// TIA Portal V17 export
// export: Created 2024-09-02T12:50:01.5701323Z, ExportSetting WithDefaults, DisplayName Totally Integrated Automation Portal, DisplayVersion V17, DisplayName TIA Portal Openness, DisplayVersion V17, DisplayName TIA Portal Version Control Interface, DisplayVersion V17, DisplayName STEP 7 Professional, DisplayVersion V17, DisplayName STEP 7 Safety, DisplayVersion V17, DisplayName WinCC Professional, DisplayVersion V17
FUNCTION_BLOCK "GraFB_Hand_51_58"   // FB1175, GRAPH
TITLE = GRAPH FB
AUTHOR : OlegFuehrus
FAMILY : SK
NAME : SK
VERSION : 0.1
// Hand functions / Handfunktionen
// stored: AcknowledgeErrorsRequired true, AutoNumber true, ExtensionBlockName LTLL_ManualGraphExt, GraphVersion 4.0, InitialValuesAcquisition false, IsIECCheckEnabled false, LanguageInNetworks LAD, LockOperatingMode false, PermanentILProcessingInMANMode true, SetENOAutomatically false, SkipSteps false, UDAEnableTagReadback false, WithAlarmHandling true
   // inherited from GRAPH_BASE
   VAR
      OFF_SQ_BASE : Bool;
   END_VAR
   VAR_INPUT
      OFF_SQ : Bool;
      INIT_SQ : Bool;
      ACK_EF : Bool;
      S_PREV : Bool;
      S_NEXT : Bool;
      SW_AUTO : Bool;
      SW_TAP : Bool;
      SW_MAN : Bool;
      S_SEL : Int;
      S_ON : Bool;
      S_OFF : Bool;
      T_PUSH : Bool;
   END_VAR
   VAR_OUTPUT
      S_NO : Int;
      S_MORE : Bool;
      S_ACTIVE : Bool;
      ERR_FLT : Bool;
      AUTO_ON : Bool;
      TAP_ON : Bool;
      MAN_ON : Bool;
   END_VAR
   VAR
      extBlock { S7_SetPoint := 'True'} : "LTLL_ManualGraphExt";
   END_VAR
   VAR_TEMP
      t_FrgHand : Bool;   // Freigabe Handbetrieb / Enable manual operation
      t_Service : Bool;   // Servicebetrieb aktiv / Service operation active
   END_VAR
BEGIN
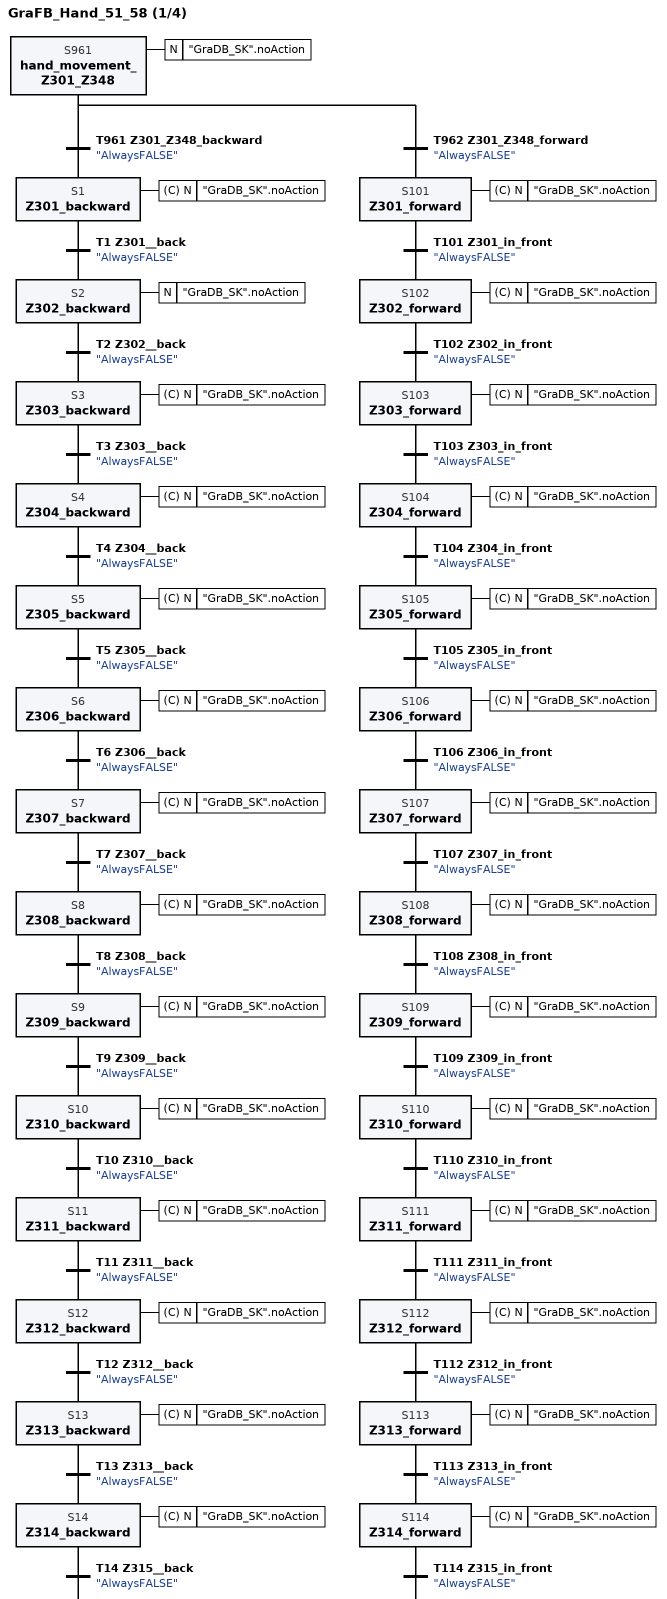
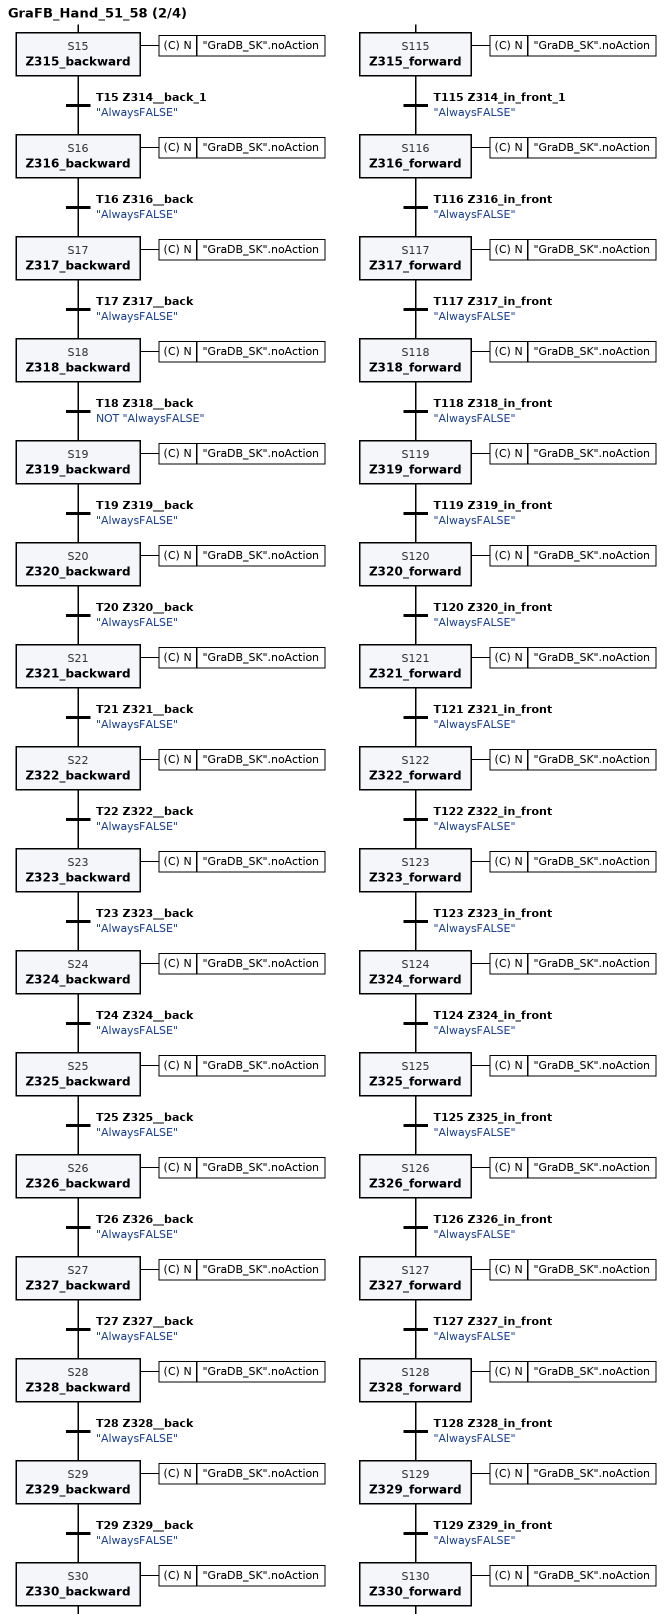
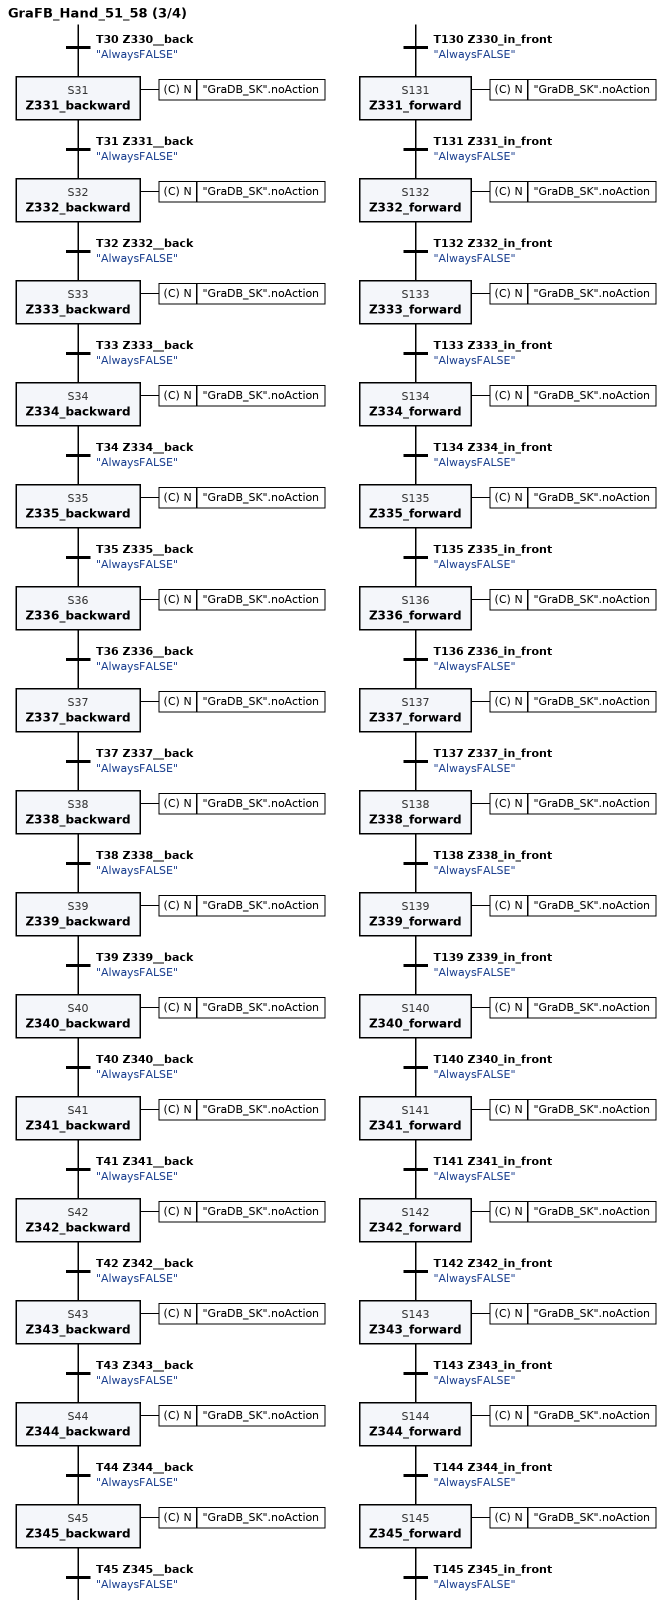
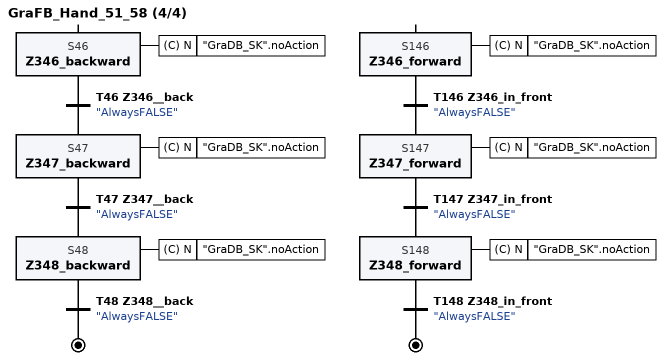
   // permanent pre-instructions
   NETWORK 1
   TITLE = HMI Lite Pass on data / HMI Lite Daten weiterreichen
      #extBlock.input := "LTLL_ManualGraphControl_OP70".screen[0].input;
   NETWORK 2
   TITLE = Instance DB Name query and pass on / Instanz DB Name abfragen und weiterreichen
      GetInstanceName(size := 0, OUT => #extBlock.input.instanceName);
   NETWORK 3
   TITLE = Interlocks Permanent machining, manual Approve and service / Interlocks Permanent Bearbeiten, Handfreigabe und Service
      IF NOT #RT_DATA.MOP.IL_PERM THEN #RT_DATA.MOP.IL_PERM := TRUE; END_IF;
      #t_FrgHand := "AnwDB_OperatingModes_OP70".BA[0]."mode_hand+start";
      #t_Service := "AnwDB_OperatingModes_OP70".BA[0].mode_service;

   // sequencer 1: Sequencer 1
   STEP hand_movement_Z301_Z348:   // S961, max time T#10S, warning time T#7S: Step commentary / Schrittkommentar
      interlock C := (none);   // hand_bereich_Z001_Z005
      supervision V := (none);   // hand_bereich_Z001_Z005
              N    "GraDB_SK".noAction
   END_STEP
   TRANSITION Z301_Z348_backward FROM hand_movement_Z301_Z348 TO Z301_backward   // T961
      := "AlwaysFALSE";
   END_TRANSITION
   TRANSITION Z301_Z348_forward FROM hand_movement_Z301_Z348 TO Z301_forward   // T962
      := "AlwaysFALSE";
   END_TRANSITION
   STEP Z301_backward:   // S1, max time T#10S, warning time T#7S
      interlock C := "AlwaysFALSE";   // Z301_zur
      supervision V := NOT #Z301__back.TT AND (#Z301_backward.T > T#5S);   // Z301_zur
      (C)     N    "GraDB_SK".noAction
   END_STEP
   TRANSITION Z301__back FROM Z301_backward TO Z302_backward   // T1
      := "AlwaysFALSE";
   END_TRANSITION
   STEP Z302_backward:   // S2, max time T#10S, warning time T#7S
      interlock C := "AlwaysFALSE";   // Z302_zur
      supervision V := NOT #Z302__back.TT AND (#Z302_backward.T > T#5S);   // Z302_zur
              N    "GraDB_SK".noAction
   END_STEP
   TRANSITION Z302__back FROM Z302_backward TO Z303_backward   // T2
      := "AlwaysFALSE";
   END_TRANSITION
   STEP Z303_backward:   // S3, max time T#10S, warning time T#7S
      interlock C := "AlwaysFALSE";   // Z303_zur
      supervision V := NOT #Z303__back.TT AND (#Z303_backward.T > T#5S);   // Z303_zur
      (C)     N    "GraDB_SK".noAction
   END_STEP
   TRANSITION Z303__back FROM Z303_backward TO Z304_backward   // T3
      := "AlwaysFALSE";
   END_TRANSITION
   STEP Z304_backward:   // S4, max time T#10S, warning time T#7S
      interlock C := "AlwaysFALSE";   // Z304_zur
      supervision V := NOT #Z304__back.TT AND (#Z304_backward.T > T#5S);   // Z304_zur
      (C)     N    "GraDB_SK".noAction
   END_STEP
   TRANSITION Z304__back FROM Z304_backward TO Z305_backward   // T4
      := "AlwaysFALSE";
   END_TRANSITION
   STEP Z305_backward:   // S5, max time T#10S, warning time T#7S
      interlock C := "AlwaysFALSE";   // Z305_zur
      supervision V := NOT #Z305__back.TT AND (#Z305_backward.T > T#5S);   // Z305_zur
      (C)     N    "GraDB_SK".noAction
   END_STEP
   TRANSITION Z305__back FROM Z305_backward TO Z306_backward   // T5
      := "AlwaysFALSE";
   END_TRANSITION
   STEP Z301_forward:   // S101, max time T#10S, warning time T#7S
      interlock C := "AlwaysFALSE";   // Z301_vor
      supervision V := NOT #Z301_in_front.TT AND (#Z301_forward.T > T#5S);   // Z301_vor
      (C)     N    "GraDB_SK".noAction
   END_STEP
   TRANSITION Z301_in_front FROM Z301_forward TO Z302_forward   // T101
      := "AlwaysFALSE";
   END_TRANSITION
   STEP Z302_forward:   // S102, max time T#10S, warning time T#7S
      interlock C := "AlwaysFALSE";   // Z302_vor
      supervision V := NOT #Z302_in_front.TT AND (#Z302_forward.T > T#5S);   // Z302_vor
      (C)     N    "GraDB_SK".noAction
   END_STEP
   TRANSITION Z302_in_front FROM Z302_forward TO Z303_forward   // T102
      := "AlwaysFALSE";
   END_TRANSITION
   STEP Z303_forward:   // S103, max time T#10S, warning time T#7S
      interlock C := "AlwaysFALSE";   // Z303_vor
      supervision V := NOT #Z303_in_front.TT AND (#Z303_forward.T > T#5S);   // Z303_vor
      (C)     N    "GraDB_SK".noAction
   END_STEP
   TRANSITION Z303_in_front FROM Z303_forward TO Z304_forward   // T103
      := "AlwaysFALSE";
   END_TRANSITION
   STEP Z304_forward:   // S104, max time T#10S, warning time T#7S
      interlock C := "AlwaysFALSE";   // Z304_vor
      supervision V := NOT #Z304_in_front.TT AND (#Z304_forward.T > T#5S);   // Z304_vor
      (C)     N    "GraDB_SK".noAction
   END_STEP
   TRANSITION Z304_in_front FROM Z304_forward TO Z305_forward   // T104
      := "AlwaysFALSE";
   END_TRANSITION
   STEP Z305_forward:   // S105, max time T#10S, warning time T#7S
      interlock C := "AlwaysFALSE";   // Z305_vor
      supervision V := NOT #Z305_in_front.TT AND (#Z305_forward.T > T#20S);   // Z305_vor
      (C)     N    "GraDB_SK".noAction
   END_STEP
   TRANSITION Z305_in_front FROM Z305_forward TO Z306_forward   // T105
      := "AlwaysFALSE";
   END_TRANSITION
   STEP Z306_backward:   // S6, max time T#10S, warning time T#7S: Cross transport 2 / Quertransport 2
      interlock C := "AlwaysFALSE";   // Z306_zur
      supervision V := NOT #Z306__back.TT AND (#Z306_backward.T > T#5S);   // Z306_zur
      (C)     N    "GraDB_SK".noAction
   END_STEP
   TRANSITION Z306__back FROM Z306_backward TO Z307_backward   // T6
      := "AlwaysFALSE";
   END_TRANSITION
   STEP Z307_backward:   // S7, max time T#10S, warning time T#7S
      interlock C := "AlwaysFALSE";   // Z307_zur
      supervision V := NOT #Z307__back.TT AND (#Z307_backward.T > T#5S);   // Z007_zur
      (C)     N    "GraDB_SK".noAction
   END_STEP
   TRANSITION Z307__back FROM Z307_backward TO Z308_backward   // T7
      := "AlwaysFALSE";
   END_TRANSITION
   STEP Z308_backward:   // S8, max time T#10S, warning time T#7S
      interlock C := "AlwaysFALSE";   // Z308_zur
      supervision V := NOT #Z308__back.TT AND (#Z308_backward.T > T#5S);   // Z308_zur
      (C)     N    "GraDB_SK".noAction
   END_STEP
   TRANSITION Z308__back FROM Z308_backward TO Z309_backward   // T8
      := "AlwaysFALSE";
   END_TRANSITION
   STEP Z309_backward:   // S9, max time T#10S, warning time T#7S
      interlock C := "AlwaysFALSE";   // Z309_zur
      supervision V := NOT #Z309__back.TT AND (#Z309_backward.T > T#5S);   // Z309_zur
      (C)     N    "GraDB_SK".noAction
   END_STEP
   TRANSITION Z309__back FROM Z309_backward TO Z310_backward   // T9
      := "AlwaysFALSE";
   END_TRANSITION
   STEP Z310_backward:   // S10, max time T#10S, warning time T#7S
      interlock C := "AlwaysFALSE";   // Z310_zur
      supervision V := NOT #Z310__back.TT AND (#Z310_backward.T > T#5S);   // Z310_zur
      (C)     N    "GraDB_SK".noAction
   END_STEP
   TRANSITION Z310__back FROM Z310_backward TO Z311_backward   // T10
      := "AlwaysFALSE";
   END_TRANSITION
   STEP Z306_forward:   // S106, max time T#10S, warning time T#7S
      interlock C := "AlwaysFALSE";   // Z306_vor
      supervision V := NOT #Z306_in_front.TT AND (#Z306_forward.T > T#5S);   // Z306_vor
      (C)     N    "GraDB_SK".noAction
   END_STEP
   TRANSITION Z306_in_front FROM Z306_forward TO Z307_forward   // T106
      := "AlwaysFALSE";
   END_TRANSITION
   STEP Z307_forward:   // S107, max time T#10S, warning time T#7S
      interlock C := "AlwaysFALSE";   // Z307_vor
      supervision V := NOT #Z307_in_front.TT AND (#Z307_forward.T > T#5S);   // Z307_vor
      (C)     N    "GraDB_SK".noAction
   END_STEP
   TRANSITION Z307_in_front FROM Z307_forward TO Z308_forward   // T107
      := "AlwaysFALSE";
   END_TRANSITION
   STEP Z308_forward:   // S108, max time T#10S, warning time T#7S
      interlock C := "AlwaysFALSE";   // Z308_vor
      supervision V := NOT #Z308_in_front.TT AND (#Z308_forward.T > T#5S);   // Z308_vor
      (C)     N    "GraDB_SK".noAction
   END_STEP
   TRANSITION Z308_in_front FROM Z308_forward TO Z309_forward   // T108
      := "AlwaysFALSE";
   END_TRANSITION
   STEP Z309_forward:   // S109, max time T#10S, warning time T#7S
      interlock C := "AlwaysFALSE";   // Z309_vor
      supervision V := NOT #Z309_in_front.TT AND (#Z309_forward.T > T#5S);   // Z309_vor
      (C)     N    "GraDB_SK".noAction
   END_STEP
   TRANSITION Z309_in_front FROM Z309_forward TO Z310_forward   // T109
      := "AlwaysFALSE";
   END_TRANSITION
   STEP Z310_forward:   // S110, max time T#10S, warning time T#7S
      interlock C := "AlwaysFALSE";   // Z310_vor
      supervision V := NOT #Z310_in_front.TT AND (#Z310_forward.T > T#5S);   // Z310_vor
      (C)     N    "GraDB_SK".noAction
   END_STEP
   TRANSITION Z310_in_front FROM Z310_forward TO Z311_forward   // T110
      := "AlwaysFALSE";
   END_TRANSITION
   STEP Z311_backward:   // S11, max time T#10S, warning time T#7S
      interlock C := "AlwaysFALSE";   // Z311_zur
      supervision V := NOT #Z311__back.TT AND (#Z311_backward.T > T#5S);   // Z311_zur
      (C)     N    "GraDB_SK".noAction
   END_STEP
   TRANSITION Z311__back FROM Z311_backward TO Z312_backward   // T11
      := "AlwaysFALSE";
   END_TRANSITION
   STEP Z312_backward:   // S12, max time T#10S, warning time T#7S
      interlock C := "AlwaysFALSE";   // Z312_zur
      supervision V := NOT #Z312__back.TT AND (#Z312_backward.T > T#5S);   // Z312_zur
      (C)     N    "GraDB_SK".noAction
   END_STEP
   TRANSITION Z312__back FROM Z312_backward TO Z313_backward   // T12
      := "AlwaysFALSE";
   END_TRANSITION
   STEP Z313_backward:   // S13, max time T#10S, warning time T#7S
      interlock C := "AlwaysFALSE";   // Z313_zur
      supervision V := NOT #Z313__back.TT AND (#Z313_backward.T > T#5S);   // Z313_zur
      (C)     N    "GraDB_SK".noAction
   END_STEP
   TRANSITION Z313__back FROM Z313_backward TO Z314_backward   // T13
      := "AlwaysFALSE";
   END_TRANSITION
   STEP Z314_backward:   // S14, max time T#10S, warning time T#7S
      interlock C := "AlwaysFALSE";   // Z314_zur
      supervision V := NOT #Z315__back.TT AND (#Z314_backward.T > T#5S);   // Z314_zur
      (C)     N    "GraDB_SK".noAction
   END_STEP
   TRANSITION Z315__back FROM Z314_backward TO Z315_backward   // T14
      := "AlwaysFALSE";
   END_TRANSITION
   STEP Z315_backward:   // S15, max time T#10S, warning time T#7S
      interlock C := "AlwaysFALSE";   // Z315_zur
      supervision V := NOT #Z316__back.TT AND (#Z315_backward.T > T#5S);   // Z315_zur
      (C)     N    "GraDB_SK".noAction
   END_STEP
   TRANSITION Z314__back_1 FROM Z315_backward TO Z316_backward   // T15
      := "AlwaysFALSE";
   END_TRANSITION
   STEP Z311_forward:   // S111, max time T#10S, warning time T#7S
      interlock C := "AlwaysFALSE";   // Z311_vor
      supervision V := NOT #Z311_in_front.TT AND (#Z311_forward.T > T#5S);   // Z311_vor
      (C)     N    "GraDB_SK".noAction
   END_STEP
   TRANSITION Z311_in_front FROM Z311_forward TO Z312_forward   // T111
      := "AlwaysFALSE";
   END_TRANSITION
   STEP Z312_forward:   // S112, max time T#10S, warning time T#7S
      interlock C := "AlwaysFALSE";   // Z312_vor
      supervision V := NOT #Z312_in_front.TT AND (#Z312_forward.T > T#5S);   // Z312_vor
      (C)     N    "GraDB_SK".noAction
   END_STEP
   TRANSITION Z312_in_front FROM Z312_forward TO Z313_forward   // T112
      := "AlwaysFALSE";
   END_TRANSITION
   STEP Z313_forward:   // S113, max time T#10S, warning time T#7S
      interlock C := "AlwaysFALSE";   // Z313_vor
      supervision V := NOT #Z313_in_front.TT AND (#Z313_forward.T > T#5S);   // Z313_vor
      (C)     N    "GraDB_SK".noAction
   END_STEP
   TRANSITION Z313_in_front FROM Z313_forward TO Z314_forward   // T113
      := "AlwaysFALSE";
   END_TRANSITION
   STEP Z314_forward:   // S114, max time T#10S, warning time T#7S
      interlock C := "AlwaysFALSE";   // Z314_vor
      supervision V := NOT #Z315_in_front.TT AND (#Z314_forward.T > T#5S);   // Z014_vor
      (C)     N    "GraDB_SK".noAction
   END_STEP
   TRANSITION Z315_in_front FROM Z314_forward TO Z315_forward   // T114
      := "AlwaysFALSE";
   END_TRANSITION
   STEP Z315_forward:   // S115, max time T#10S, warning time T#7S
      interlock C := "AlwaysFALSE";   // Z315_vor
      supervision V := NOT #Z316_in_front.TT AND (#Z315_forward.T > T#5S);   // Z315_vor
      (C)     N    "GraDB_SK".noAction
   END_STEP
   TRANSITION Z314_in_front_1 FROM Z315_forward TO Z316_forward   // T115
      := "AlwaysFALSE";
   END_TRANSITION
   STEP Z316_backward:   // S16, max time T#10S, warning time T#7S
      interlock C := "AlwaysFALSE";   // Z316_zur
      supervision V := NOT #Z316__back.TT AND (#Z316_backward.T > T#5S);   // Z316_zur
      (C)     N    "GraDB_SK".noAction
   END_STEP
   TRANSITION Z316__back FROM Z316_backward TO Z317_backward   // T16
      := "AlwaysFALSE";
   END_TRANSITION
   STEP Z317_backward:   // S17, max time T#10S, warning time T#7S
      interlock C := "AlwaysFALSE";   // Z317_zur
      supervision V := NOT #Z317__back.TT AND (#Z317_backward.T > T#5S);   // Z317_zur
      (C)     N    "GraDB_SK".noAction
   END_STEP
   TRANSITION Z317__back FROM Z317_backward TO Z318_backward   // T17
      := "AlwaysFALSE";
   END_TRANSITION
   STEP Z318_backward:   // S18, max time T#10S, warning time T#7S
      interlock C := "AlwaysFALSE";   // Z318_zur
      supervision V := NOT #Z318__back.TT AND (#Z318_backward.T > T#5S);   // Z318_zur
      (C)     N    "GraDB_SK".noAction
   END_STEP
   TRANSITION Z318__back FROM Z318_backward TO Z319_backward   // T18
      := NOT "AlwaysFALSE";
   END_TRANSITION
   STEP Z319_backward:   // S19, max time T#10S, warning time T#7S
      interlock C := "AlwaysFALSE";   // Z319_zur
      supervision V := NOT #Z319__back.TT AND (#Z319_backward.T > T#5S);   // Z319_zur
      (C)     N    "GraDB_SK".noAction
   END_STEP
   TRANSITION Z319__back FROM Z319_backward TO Z320_backward   // T19
      := "AlwaysFALSE";
   END_TRANSITION
   STEP Z320_backward:   // S20, max time T#10S, warning time T#7S
      interlock C := "AlwaysFALSE";   // Z320_zur
      supervision V := NOT #Z320__back.TT AND (#Z320_backward.T > T#5S);   // Z320_zur
      (C)     N    "GraDB_SK".noAction
   END_STEP
   TRANSITION Z320__back FROM Z320_backward TO Z321_backward   // T20
      := "AlwaysFALSE";
   END_TRANSITION
   STEP Z316_forward:   // S116, max time T#10S, warning time T#7S
      interlock C := "AlwaysFALSE";   // Z316_vor
      supervision V := NOT #Z316_in_front.TT AND (#Z316_forward.T > T#5S);   // Z316_vor
      (C)     N    "GraDB_SK".noAction
   END_STEP
   TRANSITION Z316_in_front FROM Z316_forward TO Z317_forward   // T116
      := "AlwaysFALSE";
   END_TRANSITION
   STEP Z317_forward:   // S117, max time T#10S, warning time T#7S
      interlock C := "AlwaysFALSE";   // Z317_vor
      supervision V := NOT #Z317_in_front.TT AND (#Z317_forward.T > T#5S);   // Z317_vor
      (C)     N    "GraDB_SK".noAction
   END_STEP
   TRANSITION Z317_in_front FROM Z317_forward TO Z318_forward   // T117
      := "AlwaysFALSE";
   END_TRANSITION
   STEP Z318_forward:   // S118, max time T#10S, warning time T#7S
      interlock C := "AlwaysFALSE";   // Z318_vor
      supervision V := NOT #Z318_in_front.TT AND (#Z318_forward.T > T#5S);   // Z318_vor
      (C)     N    "GraDB_SK".noAction
   END_STEP
   TRANSITION Z318_in_front FROM Z318_forward TO Z319_forward   // T118
      := "AlwaysFALSE";
   END_TRANSITION
   STEP Z319_forward:   // S119, max time T#10S, warning time T#7S
      interlock C := "AlwaysFALSE";   // Z319_vor
      supervision V := NOT #Z319_in_front.TT AND (#Z319_forward.T > T#5S);   // Z319_vor
      (C)     N    "GraDB_SK".noAction
   END_STEP
   TRANSITION Z319_in_front FROM Z319_forward TO Z320_forward   // T119
      := "AlwaysFALSE";
   END_TRANSITION
   STEP Z320_forward:   // S120, max time T#10S, warning time T#7S
      interlock C := "AlwaysFALSE";   // Z320_vor
      supervision V := NOT #Z320_in_front.TT AND (#Z320_forward.T > T#5S);   // Z320_vor
      (C)     N    "GraDB_SK".noAction
   END_STEP
   TRANSITION Z320_in_front FROM Z320_forward TO Z321_forward   // T120
      := "AlwaysFALSE";
   END_TRANSITION
   STEP Z321_backward:   // S21, max time T#10S, warning time T#7S
      interlock C := "AlwaysFALSE";   // Z321_zur
      supervision V := NOT #Z321__back.TT AND (#Z321_backward.T > T#10S);   // Z321_zur
      (C)     N    "GraDB_SK".noAction
   END_STEP
   TRANSITION Z321__back FROM Z321_backward TO Z322_backward   // T21
      := "AlwaysFALSE";
   END_TRANSITION
   STEP Z322_backward:   // S22, max time T#10S, warning time T#7S
      interlock C := "AlwaysFALSE";   // Z322_zur
      supervision V := NOT #Z322__back.TT AND (#Z322_backward.T > T#10S);   // Z322_zur
      (C)     N    "GraDB_SK".noAction
   END_STEP
   TRANSITION Z322__back FROM Z322_backward TO Z323_backward   // T22
      := "AlwaysFALSE";
   END_TRANSITION
   STEP Z323_backward:   // S23, max time T#10S, warning time T#7S
      interlock C := "AlwaysFALSE";   // Z323_zur
      supervision V := NOT #Z323__back.TT AND (#Z323_backward.T > T#10S);   // Z323_zur
      (C)     N    "GraDB_SK".noAction
   END_STEP
   TRANSITION Z323__back FROM Z323_backward TO Z324_backward   // T23
      := "AlwaysFALSE";
   END_TRANSITION
   STEP Z324_backward:   // S24, max time T#10S, warning time T#7S
      interlock C := "AlwaysFALSE";   // Z324_zur
      supervision V := NOT #Z324__back.TT AND (#Z324_backward.T > T#5S);   // Z324_zur
      (C)     N    "GraDB_SK".noAction
   END_STEP
   TRANSITION Z324__back FROM Z324_backward TO Z325_backward   // T24
      := "AlwaysFALSE";
   END_TRANSITION
   STEP Z325_backward:   // S25, max time T#10S, warning time T#7S
      interlock C := "AlwaysFALSE";   // Z325_zur
      supervision V := NOT #Z325__back.TT AND (#Z325_backward.T > T#5S);   // Z325_zur
      (C)     N    "GraDB_SK".noAction
   END_STEP
   TRANSITION Z325__back FROM Z325_backward TO Z326_backward   // T25
      := "AlwaysFALSE";
   END_TRANSITION
   STEP Z321_forward:   // S121, max time T#10S, warning time T#7S
      interlock C := "AlwaysFALSE";   // Z321_vor
      supervision V := NOT #Z321_in_front.TT AND (#Z321_forward.T > T#5S);   // Z321_vor
      (C)     N    "GraDB_SK".noAction
   END_STEP
   TRANSITION Z321_in_front FROM Z321_forward TO Z322_forward   // T121
      := "AlwaysFALSE";
   END_TRANSITION
   STEP Z322_forward:   // S122, max time T#10S, warning time T#7S
      interlock C := "AlwaysFALSE";   // Z322_vor
      supervision V := NOT #Z322_in_front.TT AND (#Z322_forward.T > T#10S);   // Z322_vor
      (C)     N    "GraDB_SK".noAction
   END_STEP
   TRANSITION Z322_in_front FROM Z322_forward TO Z323_forward   // T122
      := "AlwaysFALSE";
   END_TRANSITION
   STEP Z323_forward:   // S123, max time T#10S, warning time T#7S
      interlock C := "AlwaysFALSE";   // Z323_vor
      supervision V := NOT #Z323_in_front.TT AND (#Z323_forward.T > T#10S);   // Z323_vor
      (C)     N    "GraDB_SK".noAction
   END_STEP
   TRANSITION Z323_in_front FROM Z323_forward TO Z324_forward   // T123
      := "AlwaysFALSE";
   END_TRANSITION
   STEP Z324_forward:   // S124, max time T#10S, warning time T#7S
      interlock C := "AlwaysFALSE";   // Z324_vor
      supervision V := NOT #Z324_in_front.TT AND (#Z324_forward.T > T#5S);   // Z324_vor
      (C)     N    "GraDB_SK".noAction
   END_STEP
   TRANSITION Z324_in_front FROM Z324_forward TO Z325_forward   // T124
      := "AlwaysFALSE";
   END_TRANSITION
   STEP Z325_forward:   // S125, max time T#10S, warning time T#7S
      interlock C := "AlwaysFALSE";   // Z325_vor
      supervision V := NOT #Z325_in_front.TT AND (#Z325_forward.T > T#5S);   // Z325_vor
      (C)     N    "GraDB_SK".noAction
   END_STEP
   TRANSITION Z325_in_front FROM Z325_forward TO Z326_forward   // T125
      := "AlwaysFALSE";
   END_TRANSITION
   STEP Z326_backward:   // S26, max time T#10S, warning time T#7S
      interlock C := "AlwaysFALSE";   // Z326_zur
      supervision V := NOT #Z326__back.TT AND (#Z326_backward.T > T#5S);   // Z326_zur
      (C)     N    "GraDB_SK".noAction
   END_STEP
   TRANSITION Z326__back FROM Z326_backward TO Z327_backward   // T26
      := "AlwaysFALSE";
   END_TRANSITION
   STEP Z327_backward:   // S27, max time T#10S, warning time T#7S
      interlock C := "AlwaysFALSE";   // Z327_zur
      supervision V := NOT #Z327__back.TT AND (#Z327_backward.T > T#5S);   // Z327_zur
      (C)     N    "GraDB_SK".noAction
   END_STEP
   TRANSITION Z327__back FROM Z327_backward TO Z328_backward   // T27
      := "AlwaysFALSE";
   END_TRANSITION
   STEP Z328_backward:   // S28, max time T#10S, warning time T#7S
      interlock C := "AlwaysFALSE";   // Z328_zur
      supervision V := NOT #Z328__back.TT AND (#Z328_backward.T > T#5S);   // Z328_zur
      (C)     N    "GraDB_SK".noAction
   END_STEP
   TRANSITION Z328__back FROM Z328_backward TO Z329_backward   // T28
      := "AlwaysFALSE";
   END_TRANSITION
   STEP Z329_backward:   // S29, max time T#10S, warning time T#7S
      interlock C := "AlwaysFALSE";   // Z329_zur
      supervision V := NOT #Z329__back.TT AND (#Z329_backward.T > T#5S);   // Z329_zur
      (C)     N    "GraDB_SK".noAction
   END_STEP
   TRANSITION Z329__back FROM Z329_backward TO Z330_backward   // T29
      := "AlwaysFALSE";
   END_TRANSITION
   STEP Z330_backward:   // S30, max time T#10S, warning time T#7S
      interlock C := "AlwaysFALSE";   // Z330_zur
      supervision V := NOT #Z330__back.TT AND (#Z330_backward.T > T#5S);   // Z330_zur
      (C)     N    "GraDB_SK".noAction
   END_STEP
   TRANSITION Z330__back FROM Z330_backward TO Z331_backward   // T30
      := "AlwaysFALSE";
   END_TRANSITION
   STEP Z326_forward:   // S126, max time T#10S, warning time T#7S
      interlock C := "AlwaysFALSE";   // Z326_vor
      supervision V := NOT #Z326_in_front.TT AND (#Z326_forward.T > T#5S);   // Z326_vor
      (C)     N    "GraDB_SK".noAction
   END_STEP
   TRANSITION Z326_in_front FROM Z326_forward TO Z327_forward   // T126
      := "AlwaysFALSE";
   END_TRANSITION
   STEP Z327_forward:   // S127, max time T#10S, warning time T#7S
      interlock C := "AlwaysFALSE";   // Z327_vor
      supervision V := NOT #Z327_in_front.TT AND (#Z327_forward.T > T#5S);   // Z327_vor
      (C)     N    "GraDB_SK".noAction
   END_STEP
   TRANSITION Z327_in_front FROM Z327_forward TO Z328_forward   // T127
      := "AlwaysFALSE";
   END_TRANSITION
   STEP Z328_forward:   // S128, max time T#10S, warning time T#7S
      interlock C := "AlwaysFALSE";   // Z328_vor
      supervision V := NOT #Z328_in_front.TT AND (#Z328_forward.T > T#5S);   // Z328_vor
      (C)     N    "GraDB_SK".noAction
   END_STEP
   TRANSITION Z328_in_front FROM Z328_forward TO Z329_forward   // T128
      := "AlwaysFALSE";
   END_TRANSITION
   STEP Z329_forward:   // S129, max time T#10S, warning time T#7S
      interlock C := "AlwaysFALSE";   // Z329_vor
      supervision V := NOT #Z329_in_front.TT AND (#Z329_forward.T > T#5S);   // Z329_vor
      (C)     N    "GraDB_SK".noAction
   END_STEP
   TRANSITION Z329_in_front FROM Z329_forward TO Z330_forward   // T129
      := "AlwaysFALSE";
   END_TRANSITION
   STEP Z330_forward:   // S130, max time T#10S, warning time T#7S
      interlock C := "AlwaysFALSE";   // Z330_vor
      supervision V := NOT #Z330_in_front.TT AND (#Z330_forward.T > T#5S);   // Z330_vor
      (C)     N    "GraDB_SK".noAction
   END_STEP
   TRANSITION Z330_in_front FROM Z330_forward TO Z331_forward   // T130
      := "AlwaysFALSE";
   END_TRANSITION
   STEP Z331_backward:   // S31, max time T#10S, warning time T#7S: Step commentary / Schrittkommentar
      interlock C := "AlwaysFALSE";   // Z331_zur
      supervision V := NOT #Z331__back.TT AND (#Z331_backward.T > T#5S);   // Z331_zur
      (C)     N    "GraDB_SK".noAction
   END_STEP
   TRANSITION Z331__back FROM Z331_backward TO Z332_backward   // T31
      := "AlwaysFALSE";
   END_TRANSITION
   STEP Z332_backward:   // S32, max time T#10S, warning time T#7S: Step commentary / Schrittkommentar
      interlock C := "AlwaysFALSE";   // Z332_zur
      supervision V := NOT #Z332__back.TT AND (#Z332_backward.T > T#5S);   // Z332_zur
      (C)     N    "GraDB_SK".noAction
   END_STEP
   TRANSITION Z332__back FROM Z332_backward TO Z333_backward   // T32
      := "AlwaysFALSE";
   END_TRANSITION
   STEP Z333_backward:   // S33, max time T#10S, warning time T#7S: Step commentary / Schrittkommentar
      interlock C := "AlwaysFALSE";   // Z333_zur
      supervision V := NOT #Z333__back.TT AND (#Z333_backward.T > T#5S);   // Z333_zur
      (C)     N    "GraDB_SK".noAction
   END_STEP
   TRANSITION Z333__back FROM Z333_backward TO Z334_backward   // T33
      := "AlwaysFALSE";
   END_TRANSITION
   STEP Z334_backward:   // S34, max time T#10S, warning time T#7S: Step commentary / Schrittkommentar
      interlock C := "AlwaysFALSE";   // Z334_zur
      supervision V := NOT #Z334__back.TT AND (#Z334_backward.T > T#5S);   // Z334_zur
      (C)     N    "GraDB_SK".noAction
   END_STEP
   TRANSITION Z334__back FROM Z334_backward TO Z335_backward   // T34
      := "AlwaysFALSE";
   END_TRANSITION
   STEP Z335_backward:   // S35, max time T#10S, warning time T#7S: Step commentary / Schrittkommentar
      interlock C := "AlwaysFALSE";   // Z335_zur
      supervision V := NOT #Z335__back.TT AND (#Z335_backward.T > T#5S);   // Z335_zur
      (C)     N    "GraDB_SK".noAction
   END_STEP
   TRANSITION Z335__back FROM Z335_backward TO Z336_backward   // T35
      := "AlwaysFALSE";
   END_TRANSITION
   STEP Z331_forward:   // S131, max time T#10S, warning time T#7S: Step commentary / Schrittkommentar
      interlock C := "AlwaysFALSE";   // Z331_vor
      supervision V := NOT #Z331_in_front.TT AND (#Z331_forward.T > T#5S);   // Z331_vor
      (C)     N    "GraDB_SK".noAction
   END_STEP
   TRANSITION Z331_in_front FROM Z331_forward TO Z332_forward   // T131
      := "AlwaysFALSE";
   END_TRANSITION
   STEP Z332_forward:   // S132, max time T#10S, warning time T#7S: Step commentary / Schrittkommentar
      interlock C := "AlwaysFALSE";   // Z332_vor
      supervision V := NOT #Z332_in_front.TT AND (#Z332_forward.T > T#5S);   // Z332_vor
      (C)     N    "GraDB_SK".noAction
   END_STEP
   TRANSITION Z332_in_front FROM Z332_forward TO Z333_forward   // T132
      := "AlwaysFALSE";
   END_TRANSITION
   STEP Z333_forward:   // S133, max time T#10S, warning time T#7S: Step commentary / Schrittkommentar
      interlock C := "AlwaysFALSE";   // Z333_vor
      supervision V := NOT #Z333_in_front.TT AND (#Z333_forward.T > T#5S);   // Z333_vor
      (C)     N    "GraDB_SK".noAction
   END_STEP
   TRANSITION Z333_in_front FROM Z333_forward TO Z334_forward   // T133
      := "AlwaysFALSE";
   END_TRANSITION
   STEP Z334_forward:   // S134, max time T#10S, warning time T#7S: Step commentary / Schrittkommentar
      interlock C := "AlwaysFALSE";   // Z334_vor
      supervision V := NOT #Z334_in_front.TT AND (#Z334_forward.T > T#5S);   // Z334_vor
      (C)     N    "GraDB_SK".noAction
   END_STEP
   TRANSITION Z334_in_front FROM Z334_forward TO Z335_forward   // T134
      := "AlwaysFALSE";
   END_TRANSITION
   STEP Z335_forward:   // S135, max time T#10S, warning time T#7S: Step commentary / Schrittkommentar
      interlock C := "AlwaysFALSE";   // Z335_vor
      supervision V := NOT #Z335_in_front.TT AND (#Z335_forward.T > T#5S);   // Z335_vor
      (C)     N    "GraDB_SK".noAction
   END_STEP
   TRANSITION Z335_in_front FROM Z335_forward TO Z336_forward   // T135
      := "AlwaysFALSE";
   END_TRANSITION
   STEP Z336_backward:   // S36, max time T#10S, warning time T#7S: Step commentary / Schrittkommentar
      interlock C := "AlwaysFALSE";   // Z336_zur
      supervision V := NOT #Z336__back.TT AND (#Z336_backward.T > T#5S);   // Z336_zur
      (C)     N    "GraDB_SK".noAction
   END_STEP
   TRANSITION Z336__back FROM Z336_backward TO Z337_backward   // T36
      := "AlwaysFALSE";
   END_TRANSITION
   STEP Z337_backward:   // S37, max time T#10S, warning time T#7S: Step commentary / Schrittkommentar
      interlock C := "AlwaysFALSE";   // Z337_zur
      supervision V := NOT #Z337__back.TT AND (#Z337_backward.T > T#5S);   // Z337_zur
      (C)     N    "GraDB_SK".noAction
   END_STEP
   TRANSITION Z337__back FROM Z337_backward TO Z338_backward   // T37
      := "AlwaysFALSE";
   END_TRANSITION
   STEP Z338_backward:   // S38, max time T#10S, warning time T#7S: Step commentary / Schrittkommentar
      interlock C := "AlwaysFALSE";   // Z338_zur
      supervision V := NOT #Z338__back.TT AND (#Z338_backward.T > T#5S);   // Z338_zur
      (C)     N    "GraDB_SK".noAction
   END_STEP
   TRANSITION Z338__back FROM Z338_backward TO Z339_backward   // T38
      := "AlwaysFALSE";
   END_TRANSITION
   STEP Z339_backward:   // S39, max time T#10S, warning time T#7S: Step commentary / Schrittkommentar
      interlock C := "AlwaysFALSE";   // Z339_zur
      supervision V := NOT #Z339__back.TT AND (#Z339_backward.T > T#5S);   // Z339_zur
      (C)     N    "GraDB_SK".noAction
   END_STEP
   TRANSITION Z339__back FROM Z339_backward TO Z340_backward   // T39
      := "AlwaysFALSE";
   END_TRANSITION
   STEP Z340_backward:   // S40, max time T#10S, warning time T#7S: Step commentary / Schrittkommentar
      interlock C := "AlwaysFALSE";   // Z340_zur
      supervision V := NOT #Z340__back.TT AND (#Z340_backward.T > T#5S);   // Z340_zur
      (C)     N    "GraDB_SK".noAction
   END_STEP
   TRANSITION Z340__back FROM Z340_backward TO Z341_backward   // T40
      := "AlwaysFALSE";
   END_TRANSITION
   STEP Z336_forward:   // S136, max time T#10S, warning time T#7S: Step commentary / Schrittkommentar
      interlock C := "AlwaysFALSE";   // Z336_vor
      supervision V := NOT #Z336_in_front.TT AND (#Z336_forward.T > T#5S);   // Z336_vor
      (C)     N    "GraDB_SK".noAction
   END_STEP
   TRANSITION Z336_in_front FROM Z336_forward TO Z337_forward   // T136
      := "AlwaysFALSE";
   END_TRANSITION
   STEP Z337_forward:   // S137, max time T#10S, warning time T#7S: Step commentary / Schrittkommentar
      interlock C := "AlwaysFALSE";   // Z337_vor
      supervision V := NOT #Z337_in_front.TT AND (#Z337_forward.T > T#5S);   // Z337_vor
      (C)     N    "GraDB_SK".noAction
   END_STEP
   TRANSITION Z337_in_front FROM Z337_forward TO Z338_forward   // T137
      := "AlwaysFALSE";
   END_TRANSITION
   STEP Z338_forward:   // S138, max time T#10S, warning time T#7S: Step commentary / Schrittkommentar
      interlock C := "AlwaysFALSE";   // Z338_vor
      supervision V := NOT #Z338_in_front.TT AND (#Z338_forward.T > T#5S);   // Z338_vor
      (C)     N    "GraDB_SK".noAction
   END_STEP
   TRANSITION Z338_in_front FROM Z338_forward TO Z339_forward   // T138
      := "AlwaysFALSE";
   END_TRANSITION
   STEP Z339_forward:   // S139, max time T#10S, warning time T#7S: Step commentary / Schrittkommentar
      interlock C := "AlwaysFALSE";   // Z339_vor
      supervision V := NOT #Z339_in_front.TT AND (#Z339_forward.T > T#5S);   // Z339_vor
      (C)     N    "GraDB_SK".noAction
   END_STEP
   TRANSITION Z339_in_front FROM Z339_forward TO Z340_forward   // T139
      := "AlwaysFALSE";
   END_TRANSITION
   STEP Z340_forward:   // S140, max time T#10S, warning time T#7S: Step commentary / Schrittkommentar
      interlock C := "AlwaysFALSE";   // Z340_vor
      supervision V := NOT #Z340_in_front.TT AND (#Z340_forward.T > T#5S);   // Z340_vor
      (C)     N    "GraDB_SK".noAction
   END_STEP
   TRANSITION Z340_in_front FROM Z340_forward TO Z341_forward   // T140
      := "AlwaysFALSE";
   END_TRANSITION
   STEP Z341_backward:   // S41, max time T#10S, warning time T#7S: Step commentary / Schrittkommentar
      interlock C := "AlwaysFALSE";   // Z341_zur
      supervision V := NOT #Z341__back.TT AND (#Z341_backward.T > T#5S);   // Z341_zur
      (C)     N    "GraDB_SK".noAction
   END_STEP
   TRANSITION Z341__back FROM Z341_backward TO Z342_backward   // T41
      := "AlwaysFALSE";
   END_TRANSITION
   STEP Z342_backward:   // S42, max time T#10S, warning time T#7S: Step commentary / Schrittkommentar
      interlock C := "AlwaysFALSE";   // Z342_zur
      supervision V := NOT #Z342__back.TT AND (#Z342_backward.T > T#5S);   // Z342_zur
      (C)     N    "GraDB_SK".noAction
   END_STEP
   TRANSITION Z342__back FROM Z342_backward TO Z343_backward   // T42
      := "AlwaysFALSE";
   END_TRANSITION
   STEP Z343_backward:   // S43, max time T#10S, warning time T#7S: Step commentary / Schrittkommentar
      interlock C := "AlwaysFALSE";   // Z343_zur
      supervision V := NOT #Z343__back.TT AND (#Z343_backward.T > T#5S);   // Z343_zur
      (C)     N    "GraDB_SK".noAction
   END_STEP
   TRANSITION Z343__back FROM Z343_backward TO Z344_backward   // T43
      := "AlwaysFALSE";
   END_TRANSITION
   STEP Z344_backward:   // S44, max time T#10S, warning time T#7S: Step commentary / Schrittkommentar
      interlock C := "AlwaysFALSE";   // Z344_zur
      supervision V := NOT #Z344__back.TT AND (#Z344_backward.T > T#5S);   // Z344_zur
      (C)     N    "GraDB_SK".noAction
   END_STEP
   TRANSITION Z344__back FROM Z344_backward TO Z345_backward   // T44
      := "AlwaysFALSE";
   END_TRANSITION
   STEP Z345_backward:   // S45, max time T#10S, warning time T#7S: Step commentary / Schrittkommentar
      interlock C := "AlwaysFALSE";   // Z345_zur
      supervision V := NOT #Z345__back.TT AND (#Z345_backward.T > T#5S);   // Z045_zur
      (C)     N    "GraDB_SK".noAction
   END_STEP
   TRANSITION Z345__back FROM Z345_backward TO Z346_backward   // T45
      := "AlwaysFALSE";
   END_TRANSITION
   STEP Z341_forward:   // S141, max time T#10S, warning time T#7S
      interlock C := "AlwaysFALSE";   // Z341_vor
      supervision V := NOT #Z341_in_front.TT AND (#Z341_forward.T > T#5S);   // Z341_vor
      (C)     N    "GraDB_SK".noAction
   END_STEP
   TRANSITION Z341_in_front FROM Z341_forward TO Z342_forward   // T141
      := "AlwaysFALSE";
   END_TRANSITION
   STEP Z342_forward:   // S142, max time T#10S, warning time T#7S
      interlock C := "AlwaysFALSE";   // Z342_vor
      supervision V := NOT #Z342_in_front.TT AND (#Z342_forward.T > T#5S);   // Z342_vor
      (C)     N    "GraDB_SK".noAction
   END_STEP
   TRANSITION Z342_in_front FROM Z342_forward TO Z343_forward   // T142
      := "AlwaysFALSE";
   END_TRANSITION
   STEP Z343_forward:   // S143, max time T#10S, warning time T#7S
      interlock C := "AlwaysFALSE";   // Z343_vor
      supervision V := NOT #Z343_in_front.TT AND (#Z343_forward.T > T#5S);   // Z343_vor
      (C)     N    "GraDB_SK".noAction
   END_STEP
   TRANSITION Z343_in_front FROM Z343_forward TO Z344_forward   // T143
      := "AlwaysFALSE";
   END_TRANSITION
   STEP Z344_forward:   // S144, max time T#10S, warning time T#7S
      interlock C := "AlwaysFALSE";   // Z344_vor
      supervision V := NOT #Z344_in_front.TT AND (#Z344_forward.T > T#5S);   // Z344_vor
      (C)     N    "GraDB_SK".noAction
   END_STEP
   TRANSITION Z344_in_front FROM Z344_forward TO Z345_forward   // T144
      := "AlwaysFALSE";
   END_TRANSITION
   STEP Z345_forward:   // S145, max time T#10S, warning time T#7S
      interlock C := "AlwaysFALSE";   // Z345_vor
      supervision V := NOT #Z345_in_front.TT AND (#Z345_forward.T > T#5S);   // Z345_vor
      (C)     N    "GraDB_SK".noAction
   END_STEP
   TRANSITION Z345_in_front FROM Z345_forward TO Z346_forward   // T145
      := "AlwaysFALSE";
   END_TRANSITION
   STEP Z346_backward:   // S46, max time T#10S, warning time T#7S: Step commentary / Schrittkommentar
      interlock C := "AlwaysFALSE";   // Z346_zur
      supervision V := NOT #Z346__back.TT AND (#Z346_backward.T > T#5S);   // Z346_zur
      (C)     N    "GraDB_SK".noAction
   END_STEP
   TRANSITION Z346__back FROM Z346_backward TO Z347_backward   // T46
      := "AlwaysFALSE";
   END_TRANSITION
   STEP Z347_backward:   // S47, max time T#10S, warning time T#7S: Step commentary / Schrittkommentar
      interlock C := "AlwaysFALSE";   // Z347_zur
      supervision V := NOT #Z347__back.TT AND (#Z347_backward.T > T#5S);   // Z347_zur
      (C)     N    "GraDB_SK".noAction
   END_STEP
   TRANSITION Z347__back FROM Z347_backward TO Z348_backward   // T47
      := "AlwaysFALSE";
   END_TRANSITION
   STEP Z348_backward:   // S48, max time T#10S, warning time T#7S: Step commentary / Schrittkommentar
      interlock C := "AlwaysFALSE";   // Z348_zur
      supervision V := NOT #Z348__back.TT AND (#Z348_backward.T > T#5S);   // Z348_zur
      (C)     N    "GraDB_SK".noAction
   END_STEP
   TRANSITION Z348__back FROM Z348_backward TO END   // T48
      := "AlwaysFALSE";
   END_TRANSITION
   STEP Z346_forward:   // S146, max time T#10S, warning time T#7S: Step commentary / Schrittkommentar
      interlock C := "AlwaysFALSE";   // Z346_vor
      supervision V := NOT #Z346_in_front.TT AND (#Z346_forward.T > T#5S);   // Z346_vor
      (C)     N    "GraDB_SK".noAction
   END_STEP
   TRANSITION Z346_in_front FROM Z346_forward TO Z347_forward   // T146
      := "AlwaysFALSE";
   END_TRANSITION
   STEP Z347_forward:   // S147, max time T#10S, warning time T#7S: Step commentary / Schrittkommentar
      interlock C := "AlwaysFALSE";   // Z347_vor
      supervision V := NOT #Z347_in_front.TT AND (#Z347_forward.T > T#5S);   // Z347_vor
      (C)     N    "GraDB_SK".noAction
   END_STEP
   TRANSITION Z347_in_front FROM Z347_forward TO Z348_forward   // T147
      := "AlwaysFALSE";
   END_TRANSITION
   STEP Z348_forward:   // S148, max time T#10S, warning time T#7S: Step commentary / Schrittkommentar
      interlock C := "AlwaysFALSE";   // Z048_vor
      supervision V := NOT #Z348_in_front.TT AND (#Z348_forward.T > T#5S);   // Z048_vor
      (C)     N    "GraDB_SK".noAction
   END_STEP
   TRANSITION Z348_in_front FROM Z348_forward TO END   // T148
      := "AlwaysFALSE";
   END_TRANSITION

   // permanent post-instructions
   NETWORK 1
   TITLE = HMI Lite Pass on data / HMI Lite Daten weiterreichen
      "LTLL_ManualGraphInterlock"(ManualGraphExtOutput := #extBlock.output,
                              ManualGraphControlScreen := "LTLL_ManualGraphControl_OP70".screen[0]);
   NETWORK 2
   TITLE = Report step error / Schrittkettenfehler melden
      "SysFC_NumOfSQErrors"(FLT := #RT_DATA.SQ_FLAGS.ERR_FLT,
                            Fault_SQ := "AnwDB_OperatingModes_OP70".BA[0].error_report_SK,
                            NumOf_Fault_SQ := "AnwDB_ZP_Alarm_OP70".FaultsNoSK_ST1);
END_FUNCTION_BLOCK
